FUNCTION_BLOCK TcoDigitalSensorTests EXTENDS TcoCore._internals_TcoContext
VAR
	_signal : BOOL;
	_sut : TcoElements.TcoDigitalSensor(THIS^);
	_sutNotInitialized : TcoElements.TcoDigitalSensor(THIS^);
END_VAR

VAR
	_IsTrue_result : BOOL;	
	_IsFalse_result : BOOL;	
END_VAR

METHOD PROTECTED Main
CASE _testId OF
	50:
		_sutNotInitialized.IsTrue;
		_sutNotInitialized.IsFalse;
		_sutNotInitialized.Service();
		_sutNotInitialized.Restore();		
	100:
		_sut(inoSignal := _signal);
		_IsTrue_result :=_sut.IsTrue;		
	200:
		_sut(inoSignal := _signal);
		_IsFalse_result := _sut.IsFalse;	
END_CASE
END_METHOD

END_FUNCTION_BLOCK

(* stored: Version 1.1.0.1, ProductVersion 3.1.4024.6
   POU TcoDigitalSensorTests: Id {d9a75e6f-7650-0ec2-2a0d-3777c9193dbe}, SpecialFunc None
   Method Main: Id {3b4ad63a-c724-086e-098a-93db56db0bd9} *)
